{attribute 'qualified_only'}
{attribute 'strict'}
TYPE NciChannelType :
(
	NONE := E_ItpChannelType.ItpChannelTypeNone,
	INTERPRETER := E_ItpChannelType.ItpChannelTypeInterpreter,
	KINEMATIC := E_ItpChannelType.ItpChannelTypeKinematic,
	INVALID_ITF_VERSION := E_ItpChannelType.ItpChannelType_InvalidItfVer
) INT;
END_TYPE

(* stored: Version 1.1.0.1, ProductVersion 3.1.4024.12
   DUT NciChannelType: Id {e8df33f8-a9ee-032c-2457-afa9ef326e25} *)
